FUNCTION_BLOCK FB_HMatrix_Test EXTENDS FB_TestSuite
VAR_INPUT
END_VAR
VAR_OUTPUT
END_VAR
VAR
END_VAR

WhenSetFromComponentsExpectValuesRetained();
WhenTransformedByIdentityExpectSame();
WhenVectorTransformedExpectResult();
WhenMatrixTransformedExpectResult();

METHOD PRIVATE WhenMatrixTransformedExpectResult
VAR_INPUT
END_VAR
VAR
	H1 : HMatrix;
	H2 : HMatrix;
	H3 : HMatrix;
	R1 : RMatrix;
	V1 : Vector3;
	V2 : Vector3;
	V3 : Vector3;
	V4 : Vector3;
END_VAR
TEST('WhenMatrixTransformedExpectResult');

// @TEST-RUN
R1.SetFromAngle(PI/2,1);
V1.X := 1;
H1.SetFromComponents(R1,V1);
H2 := H1;
H3 := H1.GetTransformedHMatrix(H2);

V2.SetFromComponents(1,0,0);
V3 := H3.GetTransformedVector3(V2);
V4.SetFromComponents(0,0,-1);

// @TEST-ASSERT
AssertTrue(V3.IsNearlyEqual(V4,1E-6),'Result is not correct');

TEST_FINISHED();
END_METHOD

METHOD PRIVATE WhenSetFromComponentsExpectValuesRetained
VAR_INPUT
END_VAR
VAR
	R1 : RMatrix;
	R2 : RMatrix;
	V1 : Vector3;
	V2 : Vector3;
	H1 : HMatrix;
	H2 : HMatrix;
END_VAR
TEST('WhenSetFromComponentsExpectValuesRetained');

// @TEST-RUN
R1.SetFromAngle(PI/2,0);
V1.SetFromComponents(1,2,3);
H1.SetFromComponents(R1,V1);
H2 := H1;
H1.Clear();
R2 := H2.RMatrixComponent;
V2 := H2.Vector3Component;
// @TEST-ASSERT
AssertTrue(R1.IsEqual(R2),'Rotation component not correct');
AssertTrue(V1.IsEqual(V2),'Vector component not correct');

TEST_FINISHED();
END_METHOD

METHOD PRIVATE WhenTransformedByIdentityExpectSame
VAR_INPUT
END_VAR
VAR
	H1 : HMatrix;
	H2 : HMatrix;
	H3 : HMatrix;
	R1 : RMatrix;
	V1 : Vector3;
END_VAR
TEST('WhenTransformedByIdentityExpectSame');

// @TEST-RUN
R1.SetFromAngle(PI/2,0);
V1.SetFromComponents(1,2,3);
H1.SetFromComponents(R1,V1);
H3 := H1;
H1.TransformBy(H2);

// @TEST-ASSERT
AssertTrue(H1.IsEqual(H3),'Result is not the same');

TEST_FINISHED();
END_METHOD

METHOD PRIVATE WhenVectorTransformedExpectResult
VAR_INPUT
END_VAR
VAR
	H1 : HMatrix;
	R1 : RMatrix;
	V1 : Vector3;
	V2 : Vector3;
	V3 : Vector3;
	V4 : Vector3;
END_VAR
TEST('WhenVectorTransformedExpectResult');

// @TEST-RUN
R1.SetFromAngle(PI/2,1);//90deg rotation around Y axis
V1.X := 1;
H1.SetFromComponents(R1,V1);
V2.X := 1;
V3 := H1.GetTransformedVector3(V2);
V4.SetFromComponents(1,0,-1);

// @TEST-ASSERT
AssertTrue(V3.IsEqual(V4),'Result is not correct');

TEST_FINISHED();
END_METHOD

END_FUNCTION_BLOCK

(* stored: Version 1.1.0.1, ProductVersion 3.1.4024.9
   POU FB_HMatrix_Test: Id {8509ff9f-e6f7-466d-977b-28b12283ac53}, SpecialFunc None
   Method WhenMatrixTransformedExpectResult: Id {b9562da0-add4-4fb7-aadc-2b99f713b825}
   Method WhenSetFromComponentsExpectValuesRetained: Id {09201a71-edee-42bf-896b-1afd1555a103}
   Method WhenTransformedByIdentityExpectSame: Id {64ecb900-bfd6-4ae6-ab9e-4e9de7d0e86d}
   Method WhenVectorTransformedExpectResult: Id {0b68112b-2ff3-4256-9695-dc18fbdf33ab} *)
